(* Logix 5000 project; controller PBS_Perfusion vendor 1 type 14 code 217 rev 32.14; software revision 32.03; part 26 of 27 *)
(* tags used below, declared in another part *)
   BRX_Level_Initialize : BOOL;
   BRX_Level_Scaler : SCALE;
   CCA_3way : P_D4SD;   // TIE IO TO STATUS BITS NOT OUTPUT BITS ON p_d4sd for all 4 of them, otherwise will not hold position through power cycle
   CO2_3way : P_D4SD;
   EStop : P_DIn;
   FIC110 : P_ValveC;   // PBS CCA
   FIC110_intlk : P_Intlk;
   FIC120 : P_ValveC;   // O2 pbs
   FIC120_intlk : P_Intlk;
   FIC130 : P_ValveC;   // CO2 pbs
   FIC130_intlk : P_Intlk;
   FIC140 : P_ValveC;   // pbs N2 mfc
   FIC140_intlk : P_Intlk;
   KV111 : P_ValveSO;   // CCA Overlay Valve
   KV112 : P_ValveSO;   // CCA Sparge Valve
   KV121 : P_ValveSO;   // O2 Overlay Valve
   KV122 : P_ValveSO;   // O2 Sparge Valve
   KV131 : P_ValveSO;   // CO2 Overlay Valve
   KV132 : P_ValveSO;   // CO2 Sparge Valve
   KV141 : P_ValveSO;   // N2 Overlay Valve
   KV142 : P_ValveSO;   // N2 Sparge Valve
   Level_Control_Enable : BOOL;
   Level_Deadband_High_SP : REAL;
   Level_Deadband_Low_SP : REAL;
   LIT801 : P_AInAdv;   // Level Value From BRX
   MCV_FillWeight : REAL;
   MCV_InitialFill : BOOL;
   MCV_InitialFillRunning : BOOL;
   MCV_InitialFillSpeed : REAL;
   MCV_LoAdjTimer : TIMER;
   MCV_LoSP : REAL;
   MCV_LoTimerSP : REAL;
   MediaAdj_InProgress : BOOL;
   MediaFill_ON : BOOL;
   MediaLoSpeed : REAL;
   N2_3way : P_D4SD;
   O2_3way : P_D4SD;
   ONS : DINT[3];
   P101 : P_VSD;   // Feed Pump
   P101_Cal : Pump_Cal;
   P101_Cal_Abort : BOOL;
   P101_Cal_Accept : BOOL;
   P101_Cal_ColConst : REAL;
   P101_Cal_Collected : REAL;
   P101_Cal_Complete : BOOL;
   P101_Cal_Constant : REAL;
   P101_Cal_Max_Flow : REAL;
   P101_Cal_Running : BOOL;
   P101_Cal_Speed : REAL;   // ml/min
   p101_Cal_Start : BOOL;
   P101_Cal_Steps : REAL;
   P101_CalRevs : REAL;
   P101_Crash_Stop : AMP_Crash_Stop;
   P101_Dose_Abort : BOOL;
   P101_Dose_mL : REAL;
   P101_Dose_Running : BOOL;
   P101_Dose_Speed_mlmin : REAL;
   P101_Dose_Start : BOOL;
   P101_MaxRPM : REAL;
   P101_Motor_Constant : DINT;
   P101_Relative_Move : AMP_Relative_Move;
   P101_Speed : REAL;
   P102 : P_VSD;   // Media Pump
   P102_Cal : Pump_Cal;
   P102_Cal_Abort : BOOL;
   P102_Cal_Accept : BOOL;
   P102_Cal_ColConst : REAL;
   P102_Cal_Collected : REAL;
   P102_Cal_Complete : BOOL;
   P102_Cal_Constant : REAL;
   P102_Cal_Max_Flow : REAL;
   P102_Cal_Running : BOOL;
   P102_Cal_Speed : REAL;   // ml/min
   P102_Cal_Steps : REAL;
   P102_CalRevs : REAL;
   P102_Crash_Stop : AMP_Crash_Stop;
   P102_Dose_Abort : BOOL;
   P102_Dose_mL : REAL;
   P102_Dose_Running : BOOL;
   P102_Dose_Speed_mlmin : REAL;
   P102_Dose_Start : BOOL;
   P102_MaxRPM : REAL;
   P102_Motor_Constant : REAL;
   P102_Relative_Move : AMP_Relative_Move;
   P103 : P_VSD;   // Conditioned Media Addition Pump
   P103_Cal_Abort : BOOL;
   P103_Cal_Accept : BOOL;
   P103_Cal_ColConst : REAL;
   P103_Cal_Collected : REAL;
   P103_Cal_Complete : BOOL;
   P103_Cal_Constant : REAL;
   P103_Cal_Max_Flow : REAL;
   P103_Cal_Running : BOOL;
   P103_Cal_Speed : REAL;   // ml/min
   P103_Cal_Steps : REAL;
   P103_CalRevs : REAL;
   P103_Crash_Stop : AMP_Crash_Stop;
   P103_Dose_Abort : BOOL;
   P103_Dose_mL : REAL;
   P103_Dose_Running : BOOL;
   P103_Dose_Speed_mlmin : REAL;
   P103_Dose_Start : BOOL;
   P103_MaxRPM : REAL;
   P103_Motor_Constant : REAL;
   P103_Relative_Move : AMP_Relative_Move;
   P104 : P_VSD;   // Recirculation Pump
   P104_Cal_Abort : BOOL;
   P104_Cal_Accept : BOOL;
   P104_Cal_ColConst : REAL;
   P104_Cal_Collected : REAL;
   P104_Cal_Complete : BOOL;
   P104_Cal_Constant : REAL;
   P104_Cal_Max_Flow : REAL;
   P104_Cal_Running : BOOL;
   P104_Cal_Speed : REAL;   // ml/min
   P104_Cal_Steps : REAL;
   P104_CalRevs : REAL;
   P104_Crash_Stop : AMP_Crash_Stop;
   P104_Dose_Abort : BOOL;
   P104_Dose_mL : REAL;
   P104_Dose_Running : BOOL;
   P104_Dose_Speed_mlmin : REAL;
   P104_Dose_Start : BOOL;
   P104_MaxRPM : REAL;
   P104_Motor_Constant : REAL;
   P104_Relative_Move : AMP_Relative_Move;
   P105 : P_VSD;   // Spent Media Pump
   P105_Abort : BOOL;
   P105_DeciRPM : REAL;
   P105_Dose : REAL;   // mL
   P105_Dose_Running : BOOL;
   P105_DoseSpeed : REAL;   // mL/min
   P105_mLrev : REAL;   // mL/rev
   P105_StartDose : BOOL;
   P105_Timer : TIMER;
   Perfusion_On : BOOL;
   PlaceHolderFeedback1 : REAL;
   PlaceHolderFeedback2 : REAL;
   PlaceHolderFeedback3 : REAL;
   PlaceHolderFeedback4 : REAL;
   PlaceHolderIOFault : DINT[3];
   PlaceHolderOutput1 : REAL;
   PlaceHolderOutput2 : REAL;
   PlaceHolderOutput3 : REAL;
   PlaceHolderOutput4 : REAL;
   WT702 : P_AInAdv;   // MCV Weight
(* CM_PBS, continued *)

ROUTINE Main   (* ladder *)
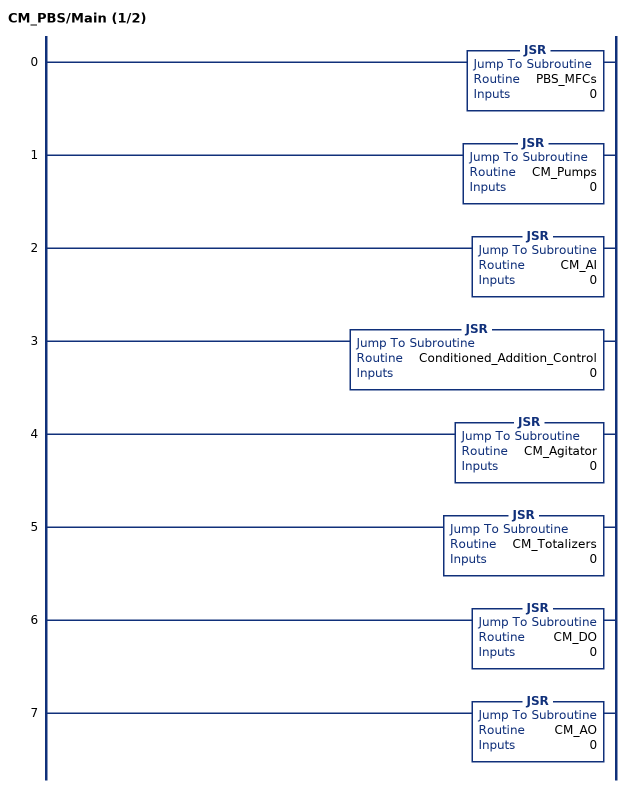
   0: JSR(PBS_MFCs,0);
   1: JSR(CM_Pumps,0);
   2: JSR(CM_AI,0);
   3: JSR(Conditioned_Addition_Control,0);
   4: JSR(CM_Agitator,0);
   5: JSR(CM_Totalizers,0);
   6: JSR(CM_DO,0);
   7: JSR(CM_AO,0);
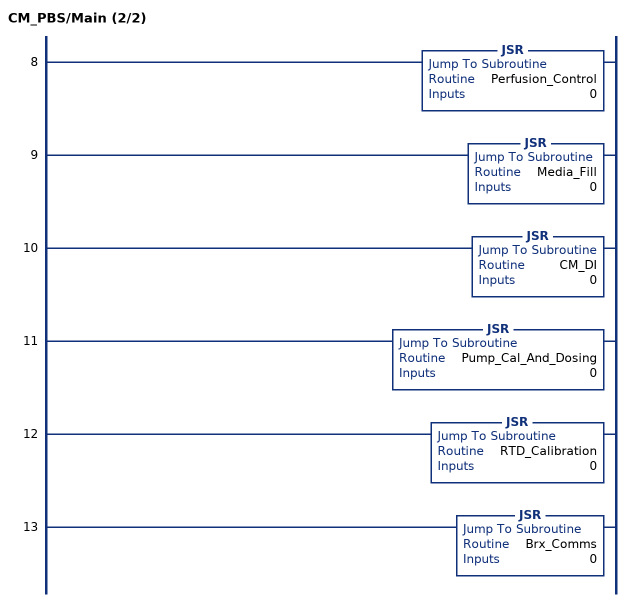
   8: JSR(Perfusion_Control,0);
   9: JSR(Media_Fill,0);
   10: JSR(CM_DI,0);
   11: JSR(Pump_Cal_And_Dosing,0);
   12: JSR(RTD_Calibration,0);
   13: JSR(Brx_Comms,0);
END_ROUTINE

ROUTINE Media_Fill   (* ladder *)
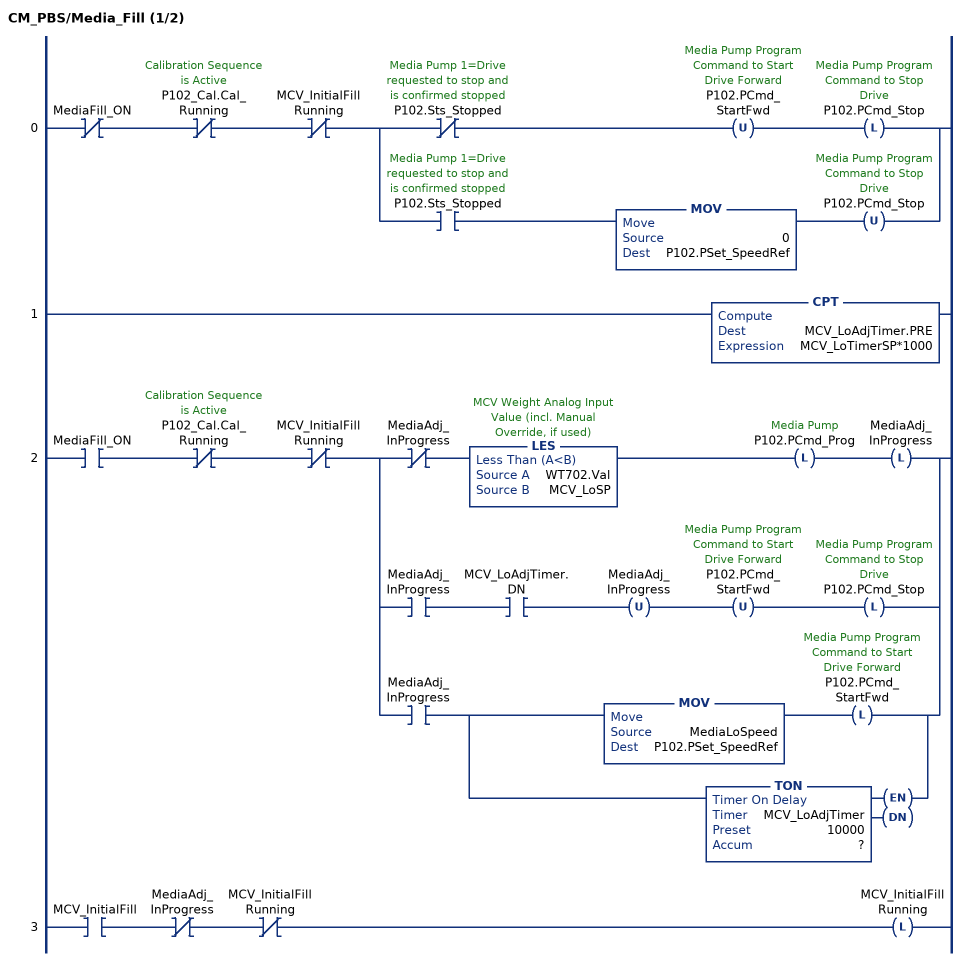
   0: XIO(MediaFill_ON)XIO(P102_Cal.Cal_Running)XIO(MCV_InitialFillRunning)[XIO(P102.Sts_Stopped) OTU(P102.PCmd_StartFwd) OTL(P102.PCmd_Stop) ,XIC(P102.Sts_Stopped) MOV(0,P102.PSet_SpeedRef) OTU(P102.PCmd_Stop) ];
   1: CPT(MCV_LoAdjTimer.PRE,MCV_LoTimerSP*1000);
   2: XIC(MediaFill_ON)XIO(P102_Cal.Cal_Running)XIO(MCV_InitialFillRunning)[XIO(MediaAdj_InProgress) LES(WT702.Val,MCV_LoSP) OTL(P102.PCmd_Prog) OTL(MediaAdj_InProgress) ,XIC(MediaAdj_InProgress) XIC(MCV_LoAdjTimer.DN) OTU(MediaAdj_InProgress) OTU(P102.PCmd_StartFwd) OTL(P102.PCmd_Stop) ,XIC(MediaAdj_InProgress) [MOV(MediaLoSpeed,P102.PSet_SpeedRef) OTL(P102.PCmd_StartFwd) ,TON(MCV_LoAdjTimer,?,?) ] ];
   3: XIC(MCV_InitialFill)XIO(MediaAdj_InProgress)XIO(MCV_InitialFillRunning)OTL(MCV_InitialFillRunning);
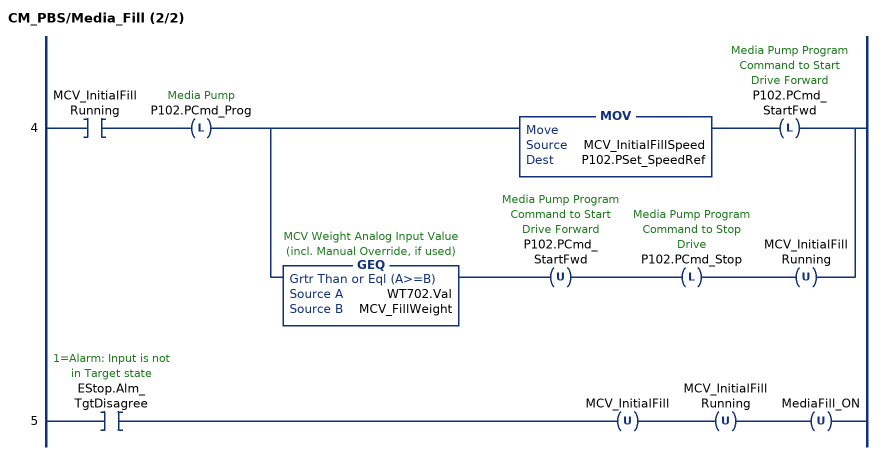
   4: XIC(MCV_InitialFillRunning)OTL(P102.PCmd_Prog)[MOV(MCV_InitialFillSpeed,P102.PSet_SpeedRef) OTL(P102.PCmd_StartFwd) ,GEQ(WT702.Val,MCV_FillWeight) OTU(P102.PCmd_StartFwd) OTL(P102.PCmd_Stop) OTU(MCV_InitialFillRunning) ];
   5: XIC(EStop.Alm_TgtDisagree)OTU(MCV_InitialFill)OTU(MCV_InitialFillRunning)OTU(MediaFill_ON);
END_ROUTINE

ROUTINE PBS_MFCs   (* ladder *)
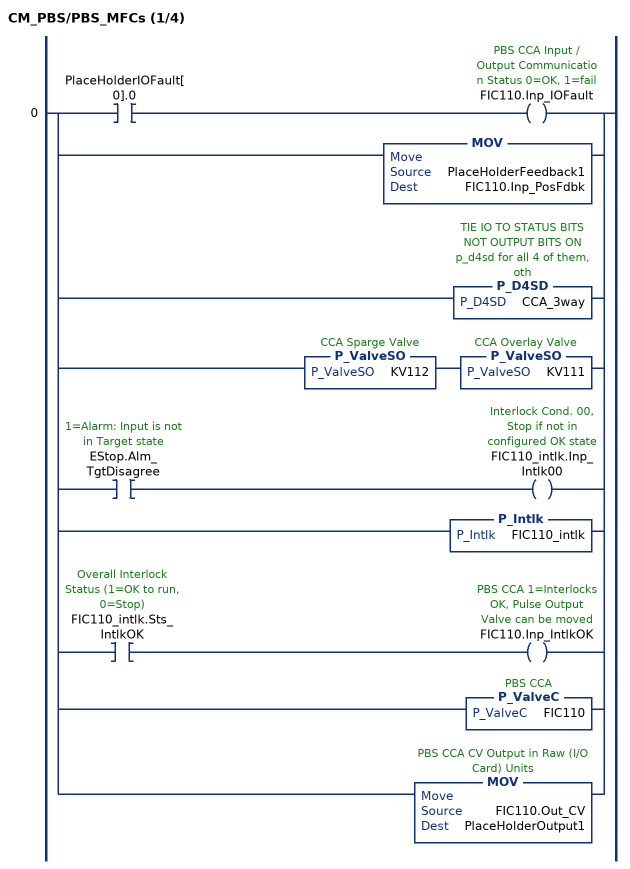
   0: [XIC(PlaceHolderIOFault[0].0) OTE(FIC110.Inp_IOFault) ,MOV(PlaceHolderFeedback1,FIC110.Inp_PosFdbk) ,P_D4SD(CCA_3way) ,P_ValveSO(KV112) P_ValveSO(KV111) ,[XIC(EStop.Alm_TgtDisagree) OTE(FIC110_intlk.Inp_Intlk00) ,P_Intlk(FIC110_intlk) ,XIC(FIC110_intlk.Sts_IntlkOK) OTE(FIC110.Inp_IntlkOK) ] ,P_ValveC(FIC110) ,MOV(FIC110.Out_CV,PlaceHolderOutput1) ];
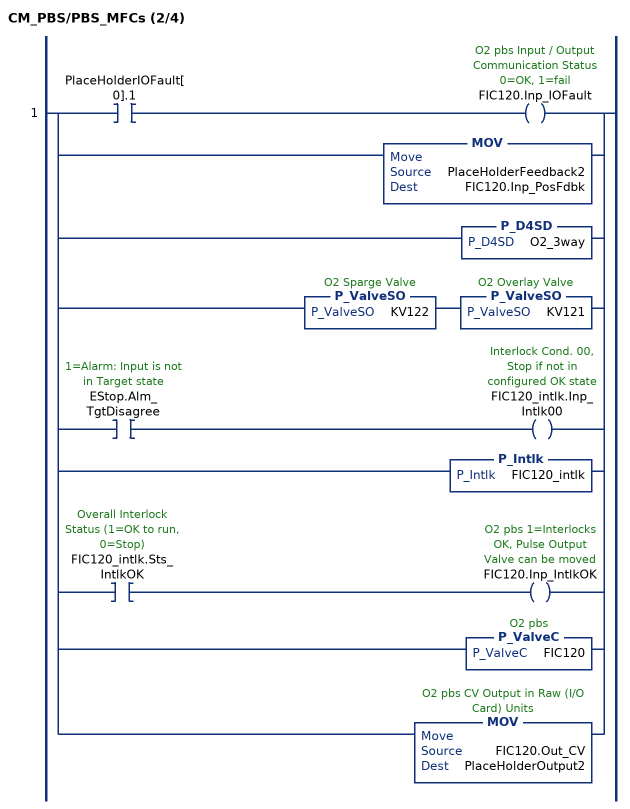
   1: [XIC(PlaceHolderIOFault[0].1) OTE(FIC120.Inp_IOFault) ,MOV(PlaceHolderFeedback2,FIC120.Inp_PosFdbk) ,P_D4SD(O2_3way) ,P_ValveSO(KV122) P_ValveSO(KV121) ,[XIC(EStop.Alm_TgtDisagree) OTE(FIC120_intlk.Inp_Intlk00) ,P_Intlk(FIC120_intlk) ,XIC(FIC120_intlk.Sts_IntlkOK) OTE(FIC120.Inp_IntlkOK) ] ,P_ValveC(FIC120) ,MOV(FIC120.Out_CV,PlaceHolderOutput2) ];
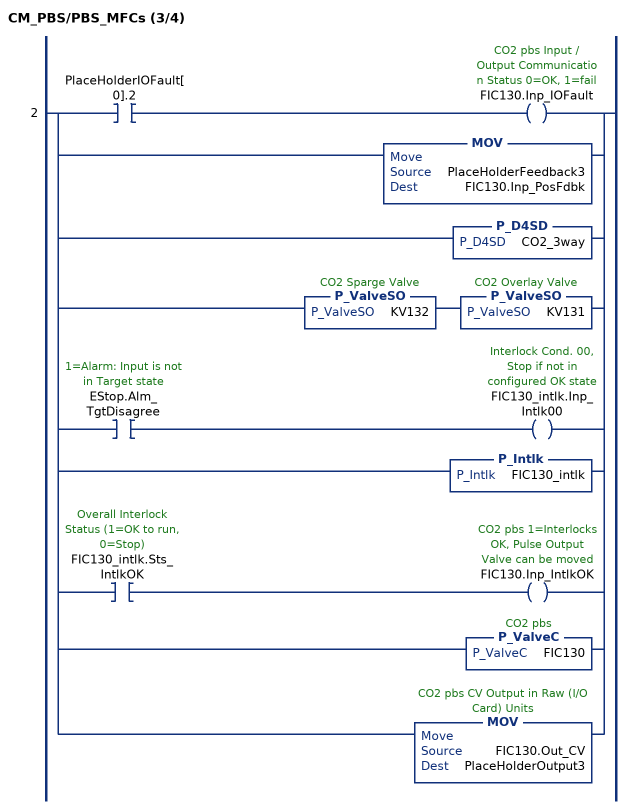
   2: [XIC(PlaceHolderIOFault[0].2) OTE(FIC130.Inp_IOFault) ,MOV(PlaceHolderFeedback3,FIC130.Inp_PosFdbk) ,P_D4SD(CO2_3way) ,P_ValveSO(KV132) P_ValveSO(KV131) ,[XIC(EStop.Alm_TgtDisagree) OTE(FIC130_intlk.Inp_Intlk00) ,P_Intlk(FIC130_intlk) ,XIC(FIC130_intlk.Sts_IntlkOK) OTE(FIC130.Inp_IntlkOK) ] ,P_ValveC(FIC130) ,MOV(FIC130.Out_CV,PlaceHolderOutput3) ];
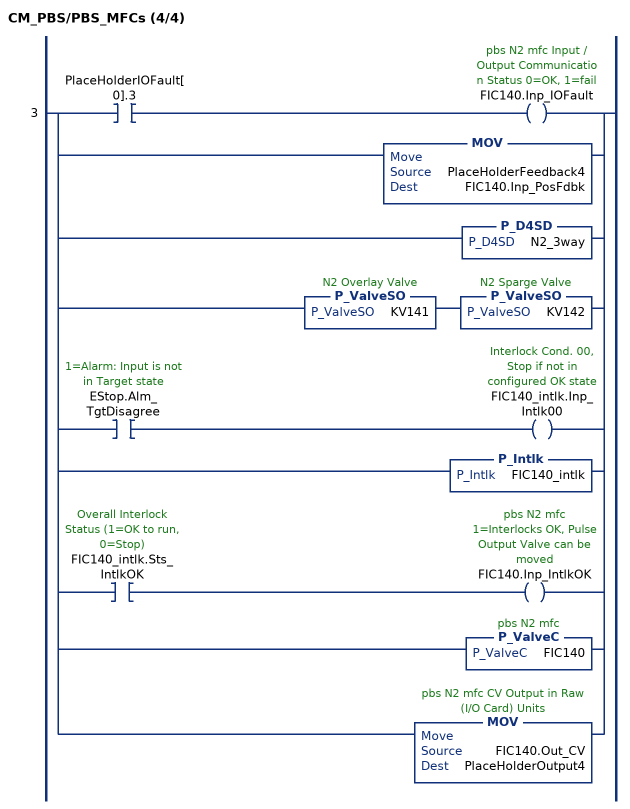
   3: [XIC(PlaceHolderIOFault[0].3) OTE(FIC140.Inp_IOFault) ,MOV(PlaceHolderFeedback4,FIC140.Inp_PosFdbk) ,P_D4SD(N2_3way) ,P_ValveSO(KV141) P_ValveSO(KV142) ,[XIC(EStop.Alm_TgtDisagree) OTE(FIC140_intlk.Inp_Intlk00) ,P_Intlk(FIC140_intlk) ,XIC(FIC140_intlk.Sts_IntlkOK) OTE(FIC140.Inp_IntlkOK) ] ,P_ValveC(FIC140) ,MOV(FIC140.Out_CV,PlaceHolderOutput4) ];
END_ROUTINE

ROUTINE Perfusion_Control   (* ladder *)
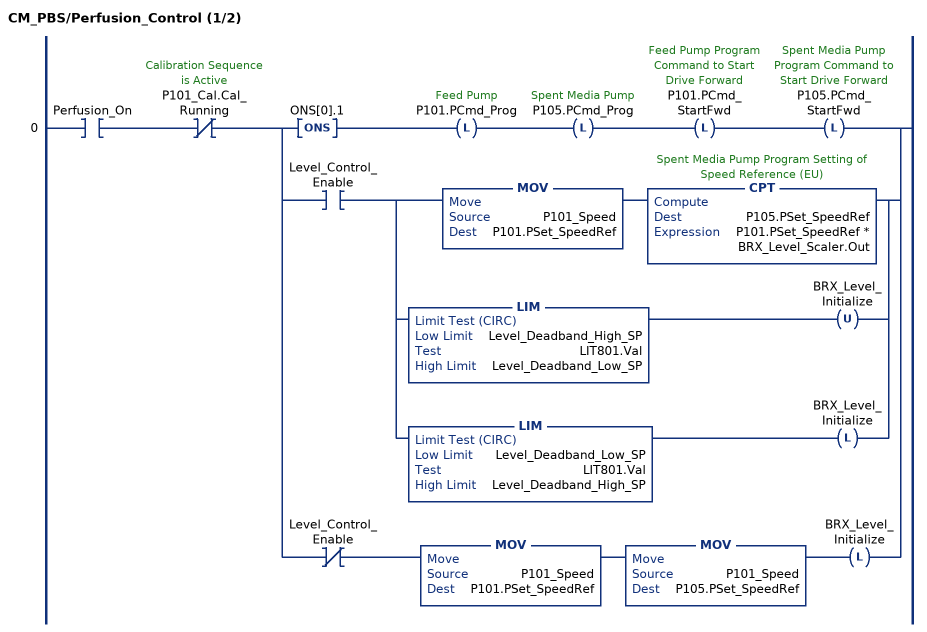
   0: XIC(Perfusion_On)XIO(P101_Cal.Cal_Running)[ONS(ONS[0].1) OTL(P101.PCmd_Prog) OTL(P105.PCmd_Prog) OTL(P101.PCmd_StartFwd) OTL(P105.PCmd_StartFwd) ,XIC(Level_Control_Enable) [MOV(P101_Speed,P101.PSet_SpeedRef) CPT(P105.PSet_SpeedRef,P101.PSet_SpeedRef * BRX_Level_Scaler.Out) ,LIM(Level_Deadband_High_SP,LIT801.Val,Level_Deadband_Low_SP) OTU(BRX_Level_Initialize) ,LIM(Level_Deadband_Low_SP,LIT801.Val,Level_Deadband_High_SP) OTL(BRX_Level_Initialize) ] ,XIO(Level_Control_Enable) MOV(P101_Speed,P101.PSet_SpeedRef) MOV(P101_Speed,P105.PSet_SpeedRef) OTL(BRX_Level_Initialize) ];
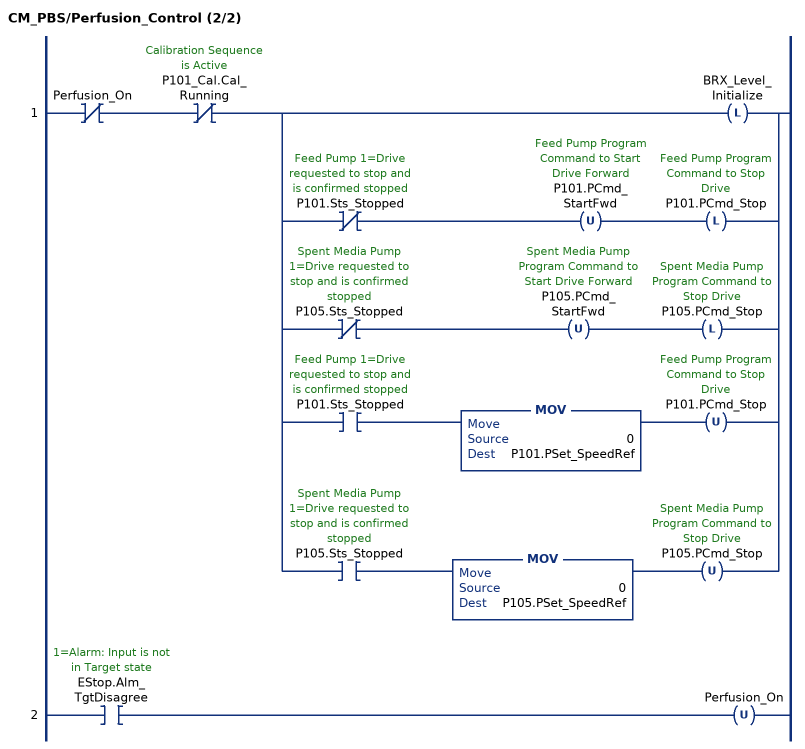
   1: XIO(Perfusion_On)XIO(P101_Cal.Cal_Running)[OTL(BRX_Level_Initialize) ,XIO(P101.Sts_Stopped) OTU(P101.PCmd_StartFwd) OTL(P101.PCmd_Stop) ,XIO(P105.Sts_Stopped) OTU(P105.PCmd_StartFwd) OTL(P105.PCmd_Stop) ,XIC(P101.Sts_Stopped) MOV(0,P101.PSet_SpeedRef) OTU(P101.PCmd_Stop) ,XIC(P105.Sts_Stopped) MOV(0,P105.PSet_SpeedRef) OTU(P105.PCmd_Stop) ];
   2: XIC(EStop.Alm_TgtDisagree)OTU(Perfusion_On);
END_ROUTINE

ROUTINE Pump_Cal_And_Dosing   (* ladder *)
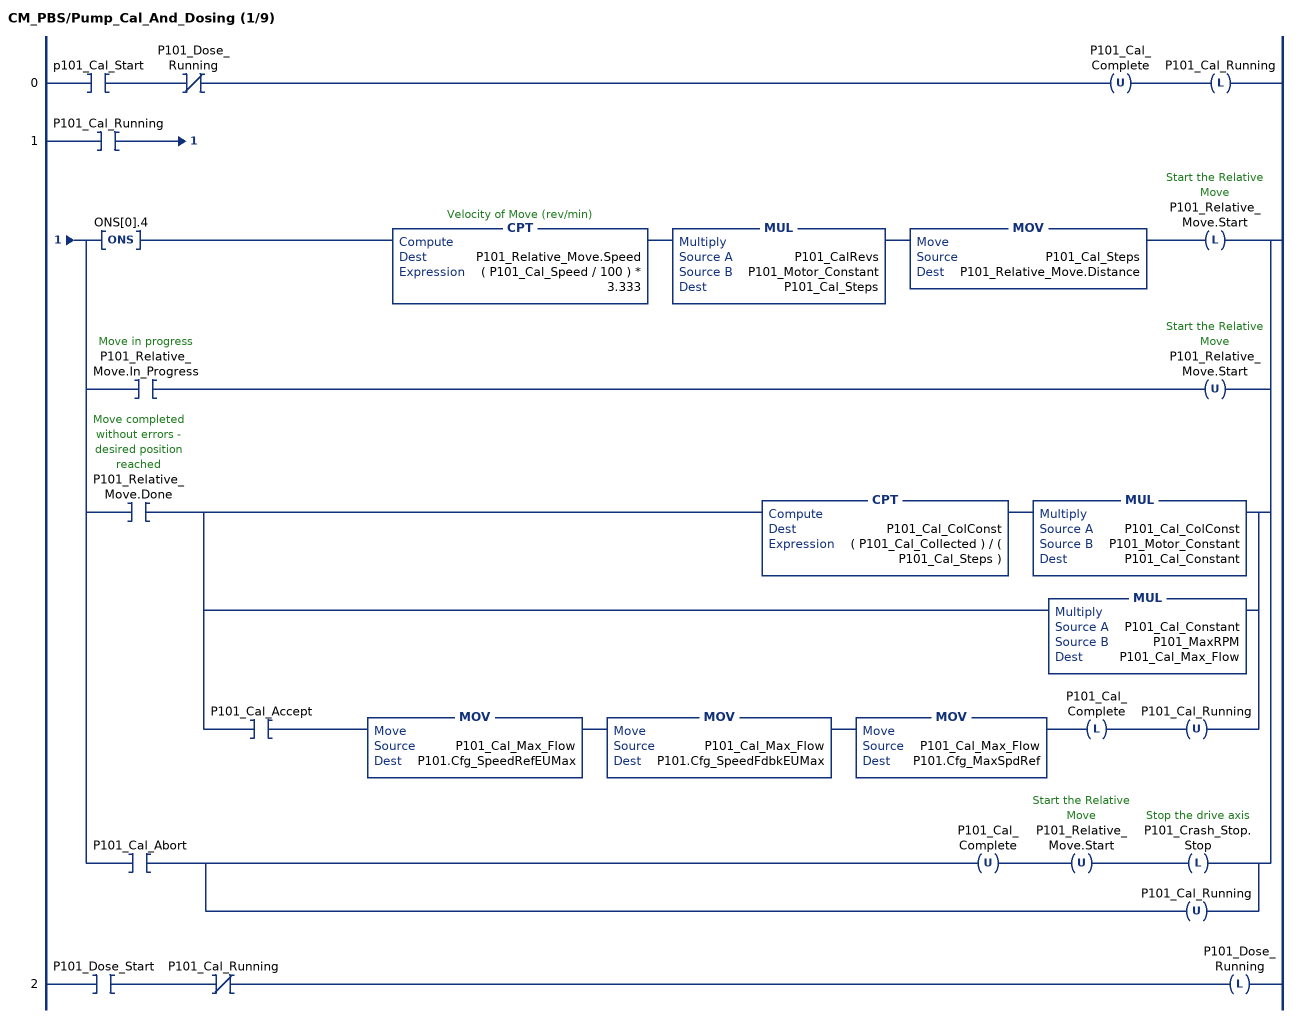
   0: XIC(p101_Cal_Start)XIO(P101_Dose_Running)OTU(P101_Cal_Complete)OTL(P101_Cal_Running);
   1: XIC(P101_Cal_Running)[ONS(ONS[0].4) CPT(P101_Relative_Move.Speed,( P101_Cal_Speed / 100 ) * 3.333) MUL(P101_CalRevs,P101_Motor_Constant,P101_Cal_Steps) MOV(P101_Cal_Steps,P101_Relative_Move.Distance) OTL(P101_Relative_Move.Start) ,XIC(P101_Relative_Move.In_Progress) OTU(P101_Relative_Move.Start) ,XIC(P101_Relative_Move.Done) [CPT(P101_Cal_ColConst,( P101_Cal_Collected ) / ( P101_Cal_Steps )) MUL(P101_Cal_ColConst,P101_Motor_Constant,P101_Cal_Constant) ,MUL(P101_Cal_Constant,P101_MaxRPM,P101_Cal_Max_Flow) ,XIC(P101_Cal_Accept) MOV(P101_Cal_Max_Flow,P101.Cfg_SpeedRefEUMax) MOV(P101_Cal_Max_Flow,P101.Cfg_SpeedFdbkEUMax) MOV(P101_Cal_Max_Flow,P101.Cfg_MaxSpdRef) OTL(P101_Cal_Complete) OTU(P101_Cal_Running) ] ,XIC(P101_Cal_Abort) [OTU(P101_Cal_Complete) OTU(P101_Relative_Move.Start) OTL(P101_Crash_Stop.Stop) ,OTU(P101_Cal_Running) ] ];
   2: XIC(P101_Dose_Start)XIO(P101_Cal_Running)OTL(P101_Dose_Running);
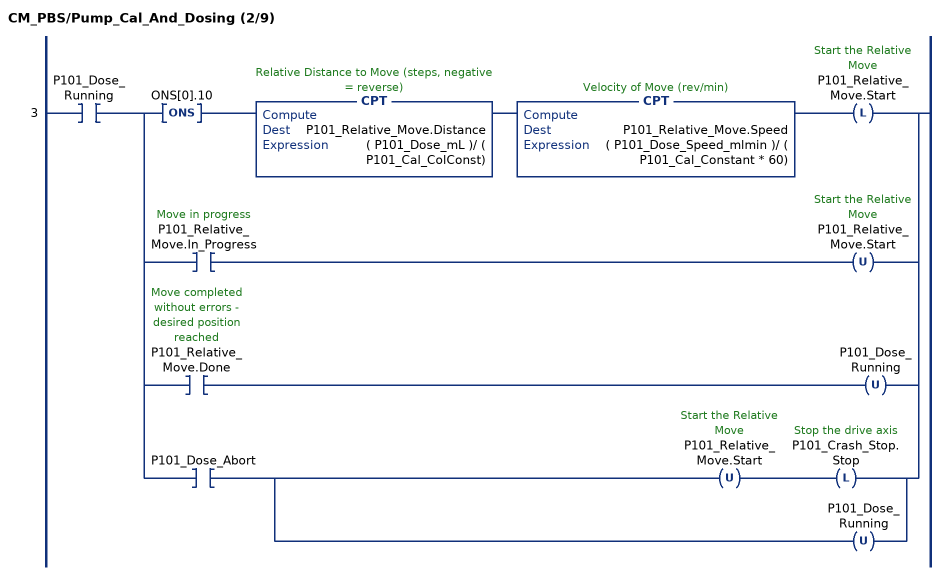
   3: XIC(P101_Dose_Running)[ONS(ONS[0].10) CPT(P101_Relative_Move.Distance,( P101_Dose_mL )/ ( P101_Cal_ColConst)) CPT(P101_Relative_Move.Speed,( P101_Dose_Speed_mlmin )/ ( P101_Cal_Constant * 60)) OTL(P101_Relative_Move.Start) ,XIC(P101_Relative_Move.In_Progress) OTU(P101_Relative_Move.Start) ,XIC(P101_Relative_Move.Done) OTU(P101_Dose_Running) ,XIC(P101_Dose_Abort) [OTU(P101_Relative_Move.Start) OTL(P101_Crash_Stop.Stop) ,OTU(P101_Dose_Running) ] ];
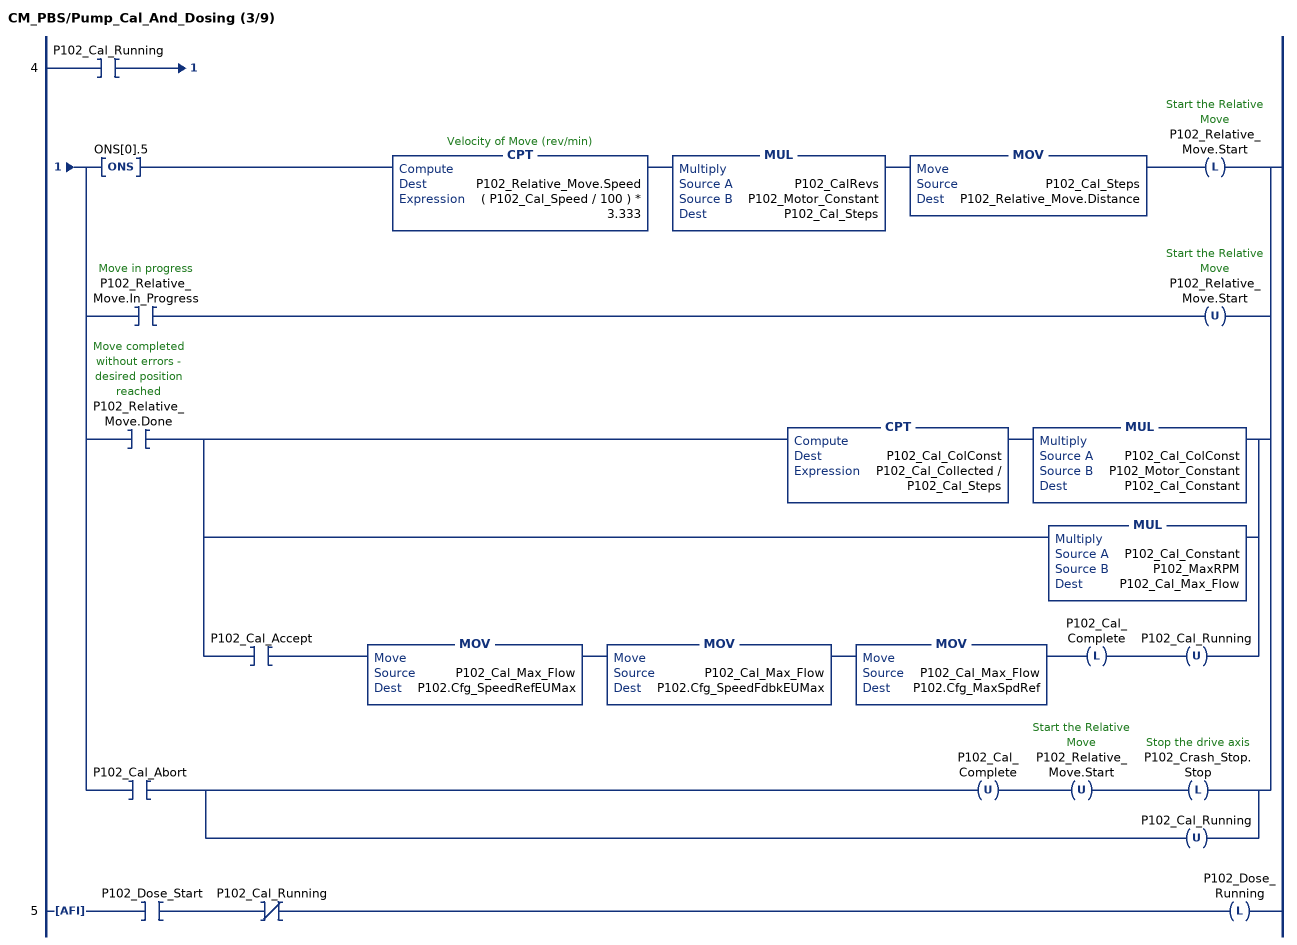
   4: XIC(P102_Cal_Running)[ONS(ONS[0].5) CPT(P102_Relative_Move.Speed,( P102_Cal_Speed / 100 ) * 3.333) MUL(P102_CalRevs,P102_Motor_Constant,P102_Cal_Steps) MOV(P102_Cal_Steps,P102_Relative_Move.Distance) OTL(P102_Relative_Move.Start) ,XIC(P102_Relative_Move.In_Progress) OTU(P102_Relative_Move.Start) ,XIC(P102_Relative_Move.Done) [CPT(P102_Cal_ColConst,P102_Cal_Collected / P102_Cal_Steps) MUL(P102_Cal_ColConst,P102_Motor_Constant,P102_Cal_Constant) ,MUL(P102_Cal_Constant,P102_MaxRPM,P102_Cal_Max_Flow) ,XIC(P102_Cal_Accept) MOV(P102_Cal_Max_Flow,P102.Cfg_SpeedRefEUMax) MOV(P102_Cal_Max_Flow,P102.Cfg_SpeedFdbkEUMax) MOV(P102_Cal_Max_Flow,P102.Cfg_MaxSpdRef) OTL(P102_Cal_Complete) OTU(P102_Cal_Running) ] ,XIC(P102_Cal_Abort) [OTU(P102_Cal_Complete) OTU(P102_Relative_Move.Start) OTL(P102_Crash_Stop.Stop) ,OTU(P102_Cal_Running) ] ];
   5: AFI()XIC(P102_Dose_Start)XIO(P102_Cal_Running)OTL(P102_Dose_Running);
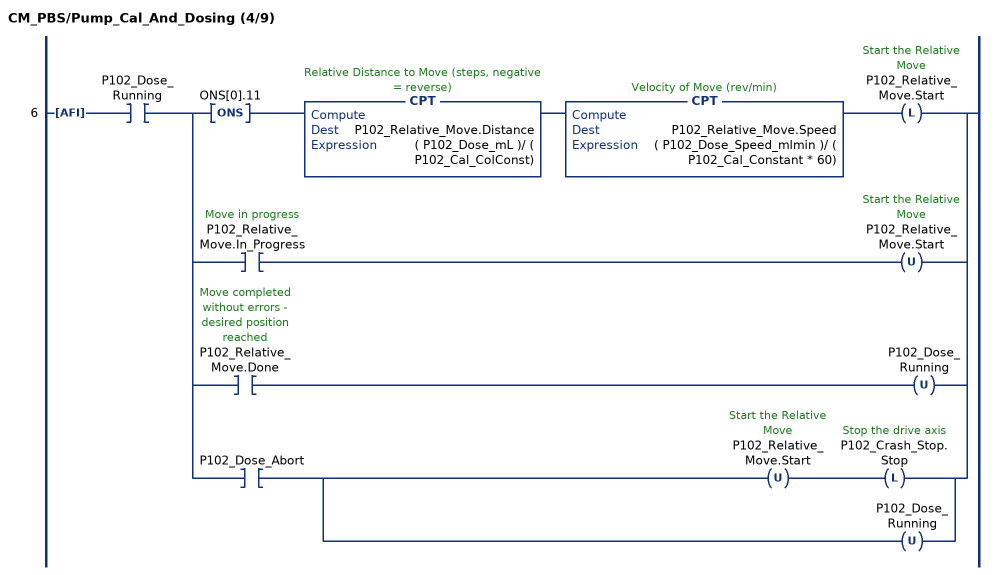
   6: AFI()XIC(P102_Dose_Running)[ONS(ONS[0].11) CPT(P102_Relative_Move.Distance,( P102_Dose_mL )/ ( P102_Cal_ColConst)) CPT(P102_Relative_Move.Speed,( P102_Dose_Speed_mlmin )/ ( P102_Cal_Constant * 60)) OTL(P102_Relative_Move.Start) ,XIC(P102_Relative_Move.In_Progress) OTU(P102_Relative_Move.Start) ,XIC(P102_Relative_Move.Done) OTU(P102_Dose_Running) ,XIC(P102_Dose_Abort) [OTU(P102_Relative_Move.Start) OTL(P102_Crash_Stop.Stop) ,OTU(P102_Dose_Running) ] ];
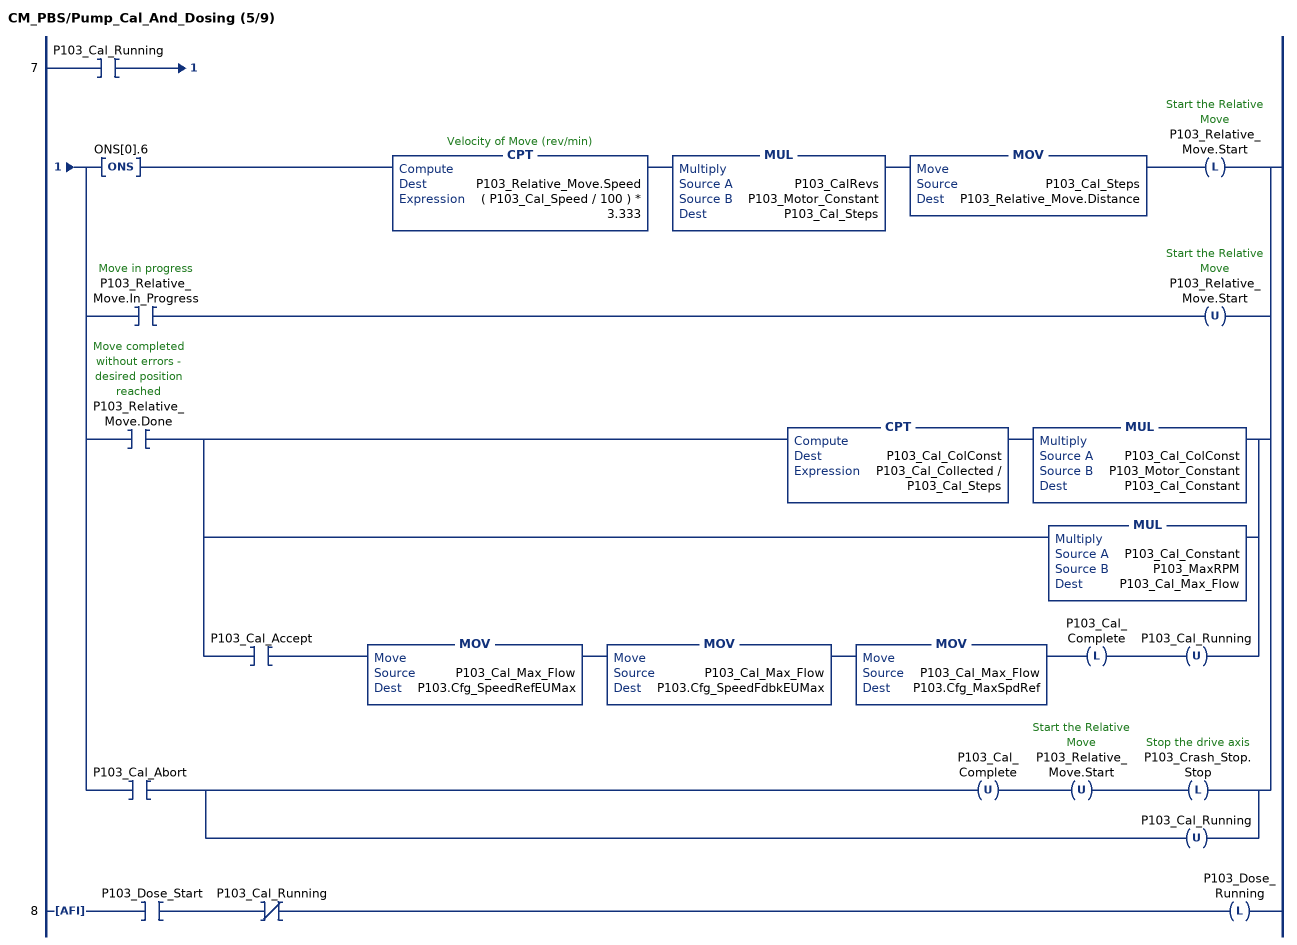
   7: XIC(P103_Cal_Running)[ONS(ONS[0].6) CPT(P103_Relative_Move.Speed,( P103_Cal_Speed / 100 ) * 3.333) MUL(P103_CalRevs,P103_Motor_Constant,P103_Cal_Steps) MOV(P103_Cal_Steps,P103_Relative_Move.Distance) OTL(P103_Relative_Move.Start) ,XIC(P103_Relative_Move.In_Progress) OTU(P103_Relative_Move.Start) ,XIC(P103_Relative_Move.Done) [CPT(P103_Cal_ColConst,P103_Cal_Collected / P103_Cal_Steps) MUL(P103_Cal_ColConst,P103_Motor_Constant,P103_Cal_Constant) ,MUL(P103_Cal_Constant,P103_MaxRPM,P103_Cal_Max_Flow) ,XIC(P103_Cal_Accept) MOV(P103_Cal_Max_Flow,P103.Cfg_SpeedRefEUMax) MOV(P103_Cal_Max_Flow,P103.Cfg_SpeedFdbkEUMax) MOV(P103_Cal_Max_Flow,P103.Cfg_MaxSpdRef) OTL(P103_Cal_Complete) OTU(P103_Cal_Running) ] ,XIC(P103_Cal_Abort) [OTU(P103_Cal_Complete) OTU(P103_Relative_Move.Start) OTL(P103_Crash_Stop.Stop) ,OTU(P103_Cal_Running) ] ];
   8: AFI()XIC(P103_Dose_Start)XIO(P103_Cal_Running)OTL(P103_Dose_Running);
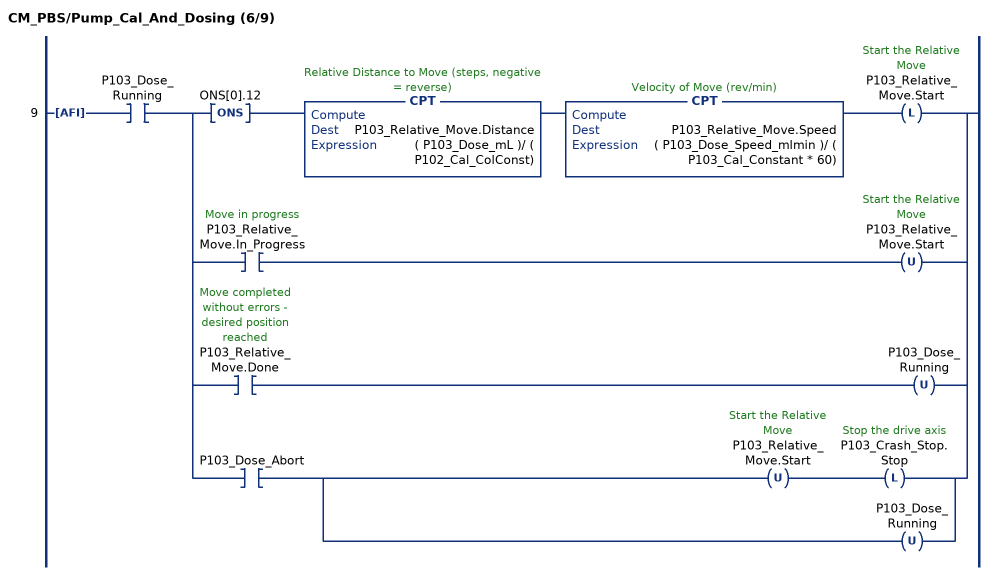
   9: AFI()XIC(P103_Dose_Running)[ONS(ONS[0].12) CPT(P103_Relative_Move.Distance,( P103_Dose_mL )/ ( P102_Cal_ColConst)) CPT(P103_Relative_Move.Speed,( P103_Dose_Speed_mlmin )/ ( P103_Cal_Constant * 60)) OTL(P103_Relative_Move.Start) ,XIC(P103_Relative_Move.In_Progress) OTU(P103_Relative_Move.Start) ,XIC(P103_Relative_Move.Done) OTU(P103_Dose_Running) ,XIC(P103_Dose_Abort) [OTU(P103_Relative_Move.Start) OTL(P103_Crash_Stop.Stop) ,OTU(P103_Dose_Running) ] ];
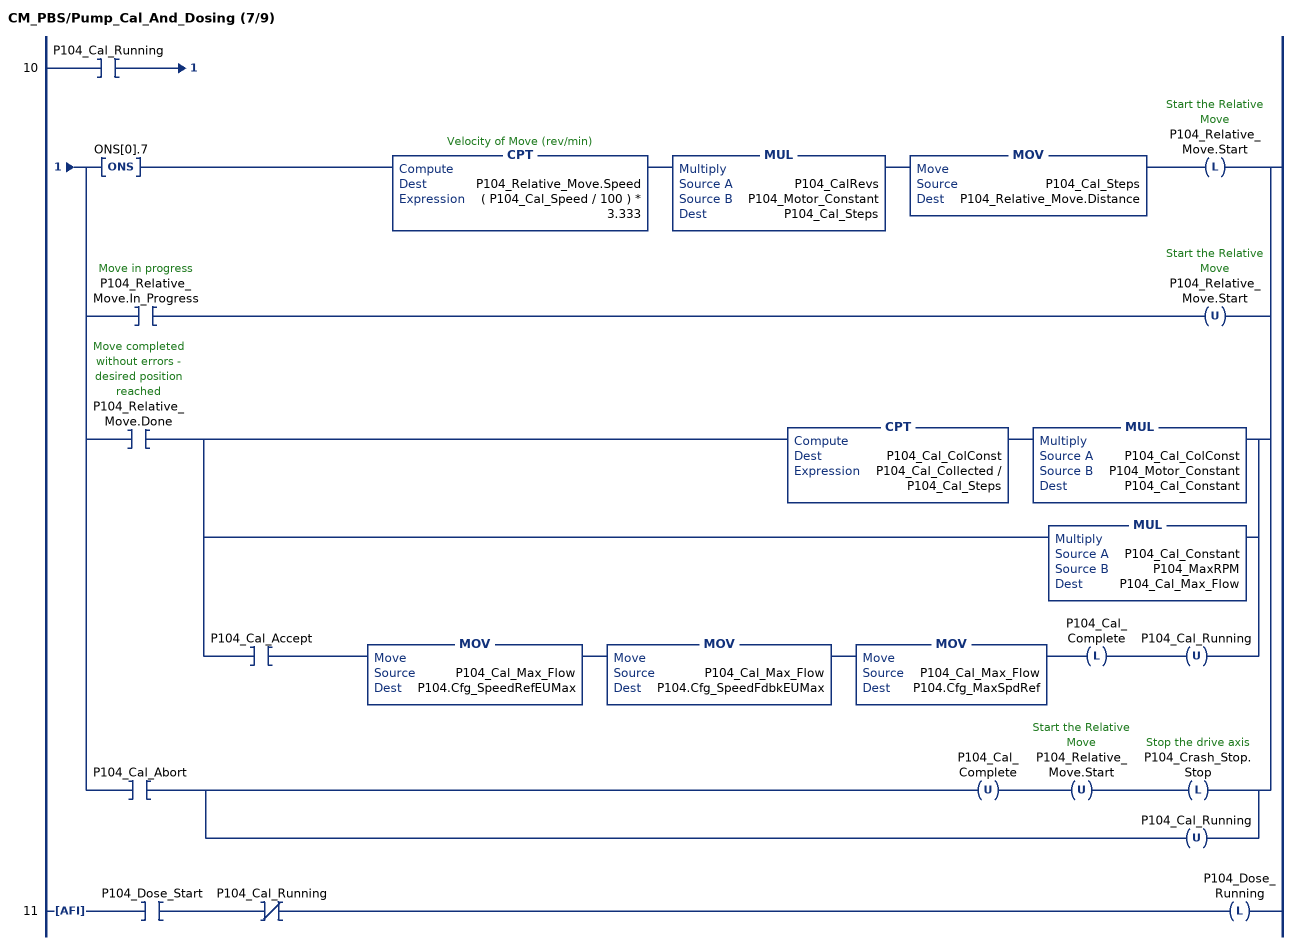
   10: XIC(P104_Cal_Running)[ONS(ONS[0].7) CPT(P104_Relative_Move.Speed,( P104_Cal_Speed / 100 ) * 3.333) MUL(P104_CalRevs,P104_Motor_Constant,P104_Cal_Steps) MOV(P104_Cal_Steps,P104_Relative_Move.Distance) OTL(P104_Relative_Move.Start) ,XIC(P104_Relative_Move.In_Progress) OTU(P104_Relative_Move.Start) ,XIC(P104_Relative_Move.Done) [CPT(P104_Cal_ColConst,P104_Cal_Collected / P104_Cal_Steps) MUL(P104_Cal_ColConst,P104_Motor_Constant,P104_Cal_Constant) ,MUL(P104_Cal_Constant,P104_MaxRPM,P104_Cal_Max_Flow) ,XIC(P104_Cal_Accept) MOV(P104_Cal_Max_Flow,P104.Cfg_SpeedRefEUMax) MOV(P104_Cal_Max_Flow,P104.Cfg_SpeedFdbkEUMax) MOV(P104_Cal_Max_Flow,P104.Cfg_MaxSpdRef) OTL(P104_Cal_Complete) OTU(P104_Cal_Running) ] ,XIC(P104_Cal_Abort) [OTU(P104_Cal_Complete) OTU(P104_Relative_Move.Start) OTL(P104_Crash_Stop.Stop) ,OTU(P104_Cal_Running) ] ];
   11: AFI()XIC(P104_Dose_Start)XIO(P104_Cal_Running)OTL(P104_Dose_Running);
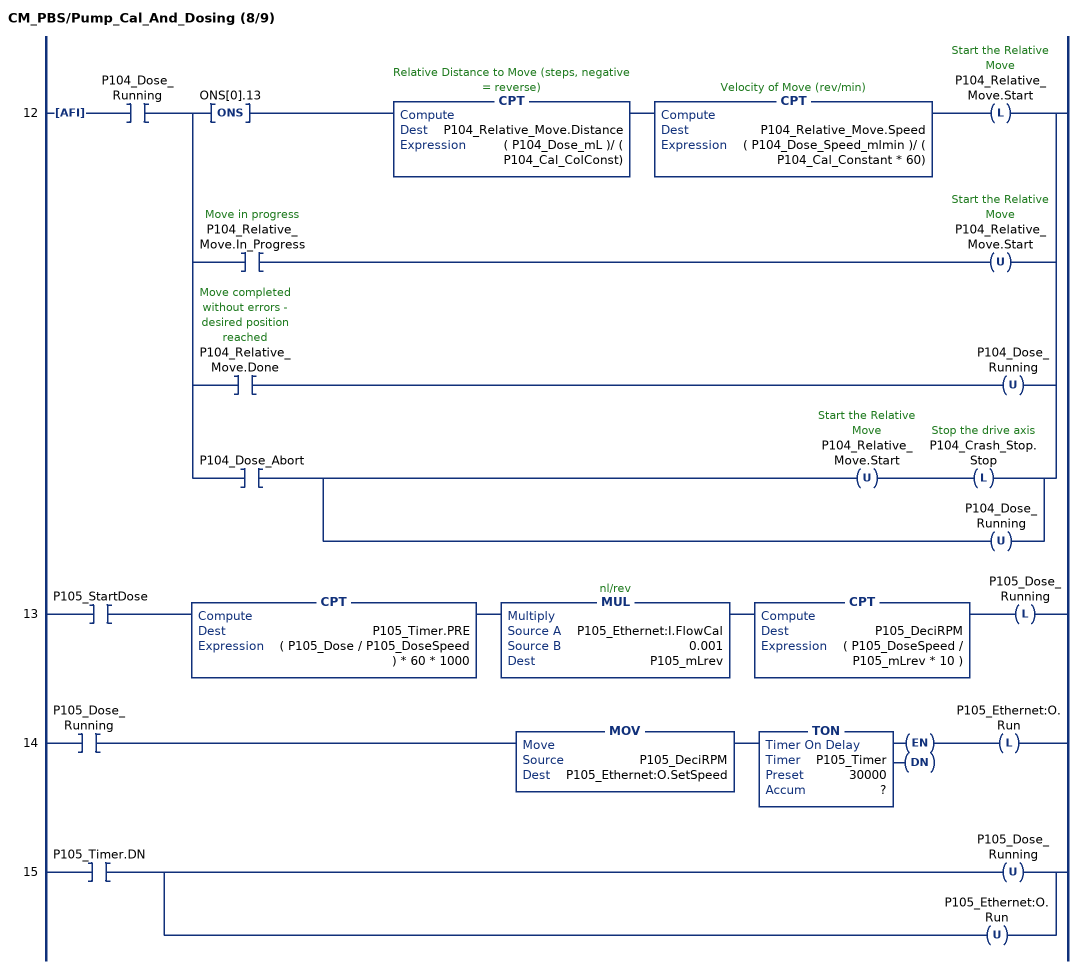
   12: AFI()XIC(P104_Dose_Running)[ONS(ONS[0].13) CPT(P104_Relative_Move.Distance,( P104_Dose_mL )/ ( P104_Cal_ColConst)) CPT(P104_Relative_Move.Speed,( P104_Dose_Speed_mlmin )/ ( P104_Cal_Constant * 60)) OTL(P104_Relative_Move.Start) ,XIC(P104_Relative_Move.In_Progress) OTU(P104_Relative_Move.Start) ,XIC(P104_Relative_Move.Done) OTU(P104_Dose_Running) ,XIC(P104_Dose_Abort) [OTU(P104_Relative_Move.Start) OTL(P104_Crash_Stop.Stop) ,OTU(P104_Dose_Running) ] ];
   13: XIC(P105_StartDose)CPT(P105_Timer.PRE,( P105_Dose / P105_DoseSpeed ) * 60 * 1000)MUL(P105_Ethernet:I.FlowCal,0.001,P105_mLrev)CPT(P105_DeciRPM,( P105_DoseSpeed / P105_mLrev * 10 ))OTL(P105_Dose_Running);
   14: XIC(P105_Dose_Running)MOV(P105_DeciRPM,P105_Ethernet:O.SetSpeed)TON(P105_Timer,?,?)OTL(P105_Ethernet:O.Run);
   15: XIC(P105_Timer.DN)[OTU(P105_Dose_Running) ,OTU(P105_Ethernet:O.Run) ];
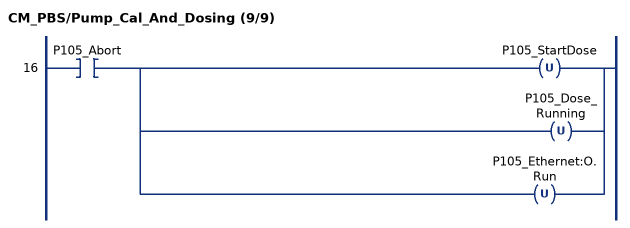
   16: XIC(P105_Abort)[OTU(P105_StartDose) ,OTU(P105_Dose_Running) ,OTU(P105_Ethernet:O.Run) ];
END_ROUTINE
